Staubli VAL3: processList.pjx

--- processList.pjx ---
Parameters version=s7.2.1 stackSize=5000 millimeterUnit=true
Program file=delete.pgx
Program file=deleteAll.pgx
Program file=getCycle.pgx
Program file=getDefaultType.pgx
Program file=getLoaded.pgx
Program file=getLoop.pgx
Program file=getPath.pgx
Program file=getSize.pgx
Program file=increase.pgx
Program file=init.pgx
Program file=insertCycle.pgx
Program file=isFound.pgx
Program file=loadProcessList.pgx
Program file=loopMode.pgx
Program file=makeFile.pgx
Program file=save.pgx
Program file=selectType.pgx
Program file=setCycle.pgx
Program file=setDefaultType.pgx
Program file=setLoop.pgx
Data file=processList.dtx
Library alias=use path=Disk://kernel/userPage/userPage.pjx
Library alias=cycleStatus path=Disk://cycleStatus/cycleStatus.pjx
Library alias=saveData path=Disk://saveData/saveData.pjx
Library alias=language path=Disk://kernel/language/language.pjx
Library alias=saveCycle path=Disk://kernel/template/session/saveCycle/saveCycle.pjx autoload=false
Library alias=prog path=Disk://instruction/PROG/PROG.pjx
Library alias=OnEvent path=Disk://OnEvent/OnEvent.pjx

--- processList.dtx ---
num nFile
string sEvent
string sProcessList
string sType
string sWrite
bool bLoading
public bool bLoop = true

--- delete.pgx ---
public program delete(num x_nIndex, num x_nType)
begin
  // mutex for the loading
  setMutex(cycleStatus:bMutex)
  switch x_nType
    case 0
      // delete a program into the process list
      logMsg("[KERNEL] CYCLE:Delete the program: "+saveCycle:sLoadStart[x_nIndex]+" at the index: "+toString("",x_nIndex))
      if size(saveCycle:sLoadStart)>1
        delete(saveCycle:sLoadStart[x_nIndex])
        delete(saveCycle:nDoneStart[x_nIndex])
        delete(saveCycle:nTotalStart[x_nIndex])
      else
        saveCycle:sLoadStart[0]=""
        saveCycle:nDoneStart[0]=0
        saveCycle:nTotalStart[0]=0
      endIf
    break
    case 1
      logMsg("[KERNEL] CYCLE:Delete the program: "+saveCycle:sLoadProg[x_nIndex]+" at the index: "+toString("",x_nIndex))
      // delete a program into the process list
      if size(saveCycle:sLoadProg)>1
        delete(saveCycle:sLoadProg[x_nIndex])
        delete(saveCycle:nDoneCycle[x_nIndex])
        delete(saveCycle:nTotalCycle[x_nIndex])
      else
        saveCycle:sLoadProg[0]=""
        saveCycle:nDoneCycle[0]=0
        saveCycle:nTotalCycle[0]=0
      endIf
    break
    case 2
      logMsg("[KERNEL] CYCLE:Delete the program: "+saveCycle:sLoadEnd[x_nIndex]+" at the index: "+toString("",x_nIndex))
      // delete a program into the process list
      if size(saveCycle:sLoadEnd)>1
        delete(saveCycle:sLoadEnd[x_nIndex])
        delete(saveCycle:nDoneEnd[x_nIndex])
        delete(saveCycle:nTotalEnd[x_nIndex])
      else
        saveCycle:sLoadEnd[0]=""
        saveCycle:nDoneEnd[0]=0
        saveCycle:nTotalEnd[0]=0
      endIf
    break
  endSwitch
//  // in order to refresh the first program
//  if x_nIndex==0
//    cycleStatus:bProgLoad=false
//    cycleStatus:sProgLoad=""
//  endIf
  //
  cycleStatus:bMutex=false
end

--- deleteAll.pgx ---
public program deleteAll(num x_nType)
  local num i
  local num nSize[3]
begin
  // onEvent
  call OnEvent:OnCycleEvent(15)
  //
  logMsg("[KERNEL] CYCLE:Delete all the program..")
  call getSize(nSize,x_nType)
  for i=0 to (nSize-1)
    call delete(0,x_nType)
  endFor
  // reinit the buffer of all the program
  // cycleStatus:bInitMemory=true
end

--- getCycle.pgx ---
public program getCycle(string& x_sName[], num& x_nTotal[], num& x_nDone[], num x_nIndex, num x_nType)
begin
  // mutex it
  // setMutex
  setMutex(cycleStatus:bMutex)
  // get the cycle from the process LIST
  switch x_nType
    case 0
      if x_nIndex<size(saveCycle:sLoadStart)
        // ON START CYCLE
        x_sName=saveCycle:sLoadStart[x_nIndex]
        x_nTotal=saveCycle:nTotalStart[x_nIndex]
        x_nDone=saveCycle:nDoneStart[x_nIndex]
      endIf
    break
    case 1
      if x_nIndex<size(saveCycle:sLoadProg)
        // get the information about the actual process list
        x_sName=saveCycle:sLoadProg[x_nIndex]
        x_nTotal=saveCycle:nTotalCycle[x_nIndex]
        x_nDone=saveCycle:nDoneCycle[x_nIndex]
      endIf
    break
    case 2
      if x_nIndex<size(saveCycle:sLoadEnd)
        // ON END CYCLE
        x_sName=saveCycle:sLoadEnd[x_nIndex]
        x_nTotal=saveCycle:nTotalEnd[x_nIndex]
        x_nDone=saveCycle:nDoneEnd[x_nIndex]
      endIf
    break
  endSwitch
  // release
  cycleStatus:bMutex=false
end

--- getDefaultType.pgx ---
public program getDefaultType(num& x_nType[])
begin
  // get the process List
  // get the last type used
  x_nType=saveCycle:nType
end

--- getLoaded.pgx ---
public program getLoaded(string& x_sLoaded[])
// get the loaded processList
begin
  // give back the actual saveCycle
  x_sLoaded=saveCycle:libPath()
  // empty the string if is the default
  if find(x_sLoaded,"template/saveCycle")!=-1
    x_sLoaded=""
  endIf
  // give back the program
  call getPath(x_sLoaded)
end

--- getLoop.pgx ---
public program getLoop(bool& x_bLoop[])
begin
  // get the loop status
  x_bLoop=saveCycle:bLoop
end

--- getPath.pgx ---
program getPath(string& x_sType[])
  local num l_nPos
  local string l_sPath
  local num i
begin
  // get the TypePath
  l_sPath=x_sType
  do
    l_nPos=find(l_sPath,"/")
    if l_nPos==-1
      l_nPos=find(l_sPath,"\")
    endIf
    if l_nPos!=-1
      l_sPath=right(l_sPath,len(l_sPath)-l_nPos-1)
    endIf
  until l_nPos==-1
  // give BACK
  x_sType=l_sPath
end

--- getSize.pgx ---
public program getSize(num& x_nSize[], num x_nType)
begin
  // get the size of the Start list
  switch x_nType
    case 0
      // get the size of the Start list
      if saveCycle:sLoadStart!=""
        x_nSize=size(saveCycle:sLoadStart)
      else
        x_nSize=0
      endIf
    break
    case 1
      if saveCycle:sLoadProg!=""
        // get the size of the process list
        x_nSize=size(saveCycle:sLoadProg)
      else
        x_nSize=0
      endIf
    break
    case 2
      if saveCycle:sLoadEnd!=""
        // get the size of the End list
        x_nSize=size(saveCycle:sLoadEnd)
      else
        x_nSize=0
      endIf
    break
  endSwitch
end

--- increase.pgx ---
public program increase(num x_nType)
begin
  // increase the size plus 1
  switch x_nType
    case 0
      // START LIST
      saveCycle:nDoneStart[cycleStatus:nProg]=saveCycle:nDoneStart[cycleStatus:nProg]+1
    break
    case 1
      // PROCESS LIST
      saveCycle:nDoneCycle[0]=saveCycle:nDoneCycle[0]+1
    break
    case 2
      // END LIST
      saveCycle:nDoneEnd[cycleStatus:nProg]=saveCycle:nDoneEnd[cycleStatus:nProg]+1
    break
  endSwitch
end

--- init.pgx ---
public program init()
  local num i
begin
  // setMutex
  setMutex(cycleStatus:bMutex)
  // START CYCLE
  for i=0 to size(saveCycle:nDoneStart)-1
    saveCycle:nDoneStart[i]=0
  endFor
  // PROCESS LIST
  if saveCycle:bLoop
    for i=0 to size(saveCycle:nDoneCycle)-1
      saveCycle:nDoneCycle[i]=0
    endFor
  endIf
  // END CYCLE
  for i=0 to size(saveCycle:nDoneEnd)-1
    saveCycle:nDoneEnd[i]=0
  endFor
  //release
  cycleStatus:bMutex=false
end

--- insertCycle.pgx ---
public program insertCycle(num x_nIndex, string x_sName, num x_nTotal, num x_nDone, num x_nType)
  local num l_nIndex
begin
  // setMutex
  setMutex(cycleStatus:bMutex)
  // insert a cycle into the process list
  //
  // use x_nIndex -1 to use FIFO politc
  //
  if x_nIndex!=-1
    l_nIndex=x_nIndex
  else
    switch x_nType
      case 0
        // start List
        if size(saveCycle:sLoadStart)==1 and saveCycle:sLoadStart[0]==""
          l_nIndex=0
        else
          l_nIndex=(size(saveCycle:sLoadStart))
        endIf
      break
      case 1
        // production list
        if size(saveCycle:sLoadProg)==1 and saveCycle:sLoadProg[0]==""
          l_nIndex=0
        else
          l_nIndex=(size(saveCycle:sLoadProg))
        endIf
      break
      case 2
        // end List
        if size(saveCycle:sLoadEnd)==1 and saveCycle:sLoadEnd[0]==""
          l_nIndex=0
        else
          l_nIndex=(size(saveCycle:sLoadEnd))
        endIf
      break
    endSwitch
  endIf
  //
  // Val3 need to have at least 1 item into a vector so...
  //
  switch x_nType
    case 0
      // ON START CYCLE
      if (l_nIndex>0) and saveCycle:sLoadStart!=""
        insert(saveCycle:sLoadStart[l_nIndex])
        insert(saveCycle:nDoneStart[l_nIndex])
        insert(saveCycle:nTotalStart[l_nIndex])
      endIf
    break
    case 1
      // get the information about the actual process list
      if (l_nIndex>0) and saveCycle:sLoadProg!=""
        insert(saveCycle:sLoadProg[l_nIndex])
        insert(saveCycle:nDoneCycle[l_nIndex])
        insert(saveCycle:nTotalCycle[l_nIndex])
      endIf
    break
    case 2
      // ON END CYCLE
      if (l_nIndex>0) and saveCycle:sLoadEnd!=""
        insert(saveCycle:sLoadEnd[l_nIndex])
        insert(saveCycle:nDoneEnd[l_nIndex])
        insert(saveCycle:nTotalEnd[l_nIndex])
      endIf
    break
  endSwitch
  // set the cycle
  call setCycle(x_sName,x_nTotal,x_nDone,l_nIndex,x_nType)
  //release
  cycleStatus:bMutex=false
end

--- isFound.pgx ---
public program isFound(string& x_sName[], bool& x_bFound[])
  local num i
  local num j
  local num l_nSize[3]
  local string l_sString
  local num k
  local num l_nResult
  local string l_sEmpty
  local num l_nID
begin
  //
  // find if a program is inside the processList
  //
  x_bFound=false
  //
  // update
  //
  l_sEmpty=""
  call use:stringCopy(l_sEmpty,sProcessList)
  // check all
  call loadProcessList(l_nResult)
  // get the size of the three processList
  for i=0 to 2
    call getSize(l_nSize[i],i)
    // look in all the program
    for j=0 to max(l_nSize[i]-1,0)
      l_nID=0
      call getCycle(l_sString,l_nID,l_nID,j,i)
      if l_sString==x_sName
        x_bFound=true
        x_sName=l_sString
        return
      endIf
    endFor
  endFor
end

--- loadProcessList.pgx ---
public program loadProcessList(num& x_nResult[])
// load the process list
  local num i
  local string l_sMessage
  local string l_sMessage2
begin
  // setMutex
  setMutex(cycleStatus:bMutex)
  // load a different processList
  if cycleStatus:bCycle==false and cycleStatus:bSimulation==false
    //saveData:sPathPList+x_sProcess
    x_nResult=saveCycle:libLoad(saveData:sPathPList)
    delay(0)
    if saveData:bDebug and x_nResult!=0
      logMsg("[KERNEL] SETPROCESSLIST:Loading processList, CODE: "+toString("",x_nResult))
    endIf
    // check the result
    if x_nResult!=0
      // load the template and empty the list
      x_nResult=saveCycle:libLoad("kernel/template/session/saveCycle")
      delay(0)
      libDelete(saveData:sPathPList)
      saveCycle:libSave(saveData:sPathPList)
      // default process list has been charged
      call language:message(l_sMessage,-7)
      call language:message(l_sMessage2,97)
      popUpMsg(l_sMessage+"saveCycle... "+l_sMessage2)
    endIf
  else
    x_nResult=-1
  endIf
  //release
  cycleStatus:bMutex=false
end

--- loopMode.pgx ---
public program loopMode()
  local num i
  local string sSwapLoad
  local num nSwapTotal
  local num l_nSize
begin
  //  set the process list after one cycle done
  //
  //  the variable loadProg has to not be minus than 1 items
  //  THIS IS THE NO LOOP CODE
  //
  if !saveCycle:bLoop
    //
    call delete(0,1)
  else
    //
    //  LOOP MODE
    //
    call getSize(l_nSize,1)
    if cycleStatus:nProg<l_nSize-1
      // continue
      cycleStatus:nProg=cycleStatus:nProg+1
    else
      // REINIT
      for i=0 to l_nSize-1
        saveCycle:nDoneCycle[i]=0
      endFor
      cycleStatus:nProg=0
    endIf
  endIf
end

--- makeFile.pgx ---
public program makeFile()
  local num i
  local num j
  local num l_nSize[3]
  local num l_nType
  local string l_sProg
  local string l_sFill
  local string l_sMessage
  local string l_sEmpty
  local num l_nID
begin
  // check if the cycle is not running
  if cycleStatus:bCycle==false and cycleStatus:bSimulation==false
    // scan all the processList
    for i=0 to 2
      call getSize(l_nSize[i],i)
    endFor
    // check if the process List is empty
    if l_nSize[1]==0
      // show message
      call language:message(l_sMessage,91)
      popUpMsg(l_sMessage)
      // came back
      return
    endIf
    // scan it
    for l_nType=0 to 2
      //
      // init
      l_sEmpty=""
      call use:stringCopy(l_sEmpty,prog:sWrite)
      //
      switch l_nType
        case 0
          // START PROCESS LIST
          // open the file
          nFile=$fileOpen("start.txt","w")
        break
        case 1
          // PROCESS LIST
          // open the file
          nFile=$fileOpen("production.txt","w")
        break
        case 2
          // END PROCESS LIST
          // open the file
          nFile=$fileOpen("end.txt","w")
        break
      endSwitch
      // scan all the program
      if l_nSize[l_nType]>0
        for i=0 to (l_nSize[l_nType]-1)
          // get the cycle
          l_nID=0
          call getCycle(l_sProg,l_nID,l_nID,i,l_nType)
          // scan the system and save the process List
          // add the program name
          insert(prog:sWrite[0])
          insert(prog:sWrite[0])
          insert(prog:sWrite[0])
          // insert the program NAME
          for j=0 to len(l_sProg)-1
            l_sFill=l_sFill+"═"
          endFor
          prog:sWrite[0]="╔═════"+l_sFill+"╗"
          prog:sWrite[1]="║PROG "+l_sProg+"║"
          prog:sWrite[2]="╚═════"+l_sFill+"╝"
          // scan the program
          call use:timerDialog("Scanning the program: "+l_sProg+"# please wait...",0)
          l_nID=3
          call prog:scanning(l_sProg,0,l_nID,true)
          // write to the file
          $fileSet(nFile,prog:sWrite,size(prog:sWrite))
          // reset the sWrite buffer
          l_sEmpty=""
          call use:stringCopy(l_sEmpty,prog:sWrite)
          l_sFill=""
        endFor
        // save the file
        $fileClose(nFile)
      endIf
    endFor
  endIf
end

--- save.pgx ---
public program save()
// save the process list
  local num i
begin
  // setMutex
  setMutex(cycleStatus:bMutex)
  // save IT
  if saveCycle:libSave()!=0
    delay(0.5)
    i=saveCycle:libSave()
    if i!=0
      popUpMsg("libsave cycle error: "+toString("",i))
      logMsg("[KERNEL] CYCLE:Error saving cycle "+toString("",i))
    endIf
  endIf
  //release
  cycleStatus:bMutex=false
end

--- selectType.pgx ---
public program selectType()
  local string l_sMessage
  local num l_nIndex
  local string l_sEvent
  local num l_nDefault
  local num l_nKey
  local num i
begin
  // select the type of the process LIST
  call use:clear(0,13)
  call language:message(l_sMessage,191)
  call use:typeCenter(13,l_sMessage,40,true)
  call use:setSizeList(10,2,15,6)
  // TODO message
  call use:listcreate("")
  call use:listadd(sType)
  call getDefaultType(l_nDefault)
  call use:selectNewField(l_nDefault,0,0)
  // select the Item
  do
    l_nKey=get()
    call use:listevent(l_nKey,l_nIndex,l_sEvent)
    // search for a key
  until l_nKey==270 or l_nKey==255
  if l_nKey==270
    call setDefaultType(l_nIndex)
    use:bUseRefresh=true
  endIf
  //
end

--- setCycle.pgx ---
public program setCycle(string x_sName, num x_nTotal, num x_nDone, num x_nIndex, num x_nType)
begin
  // insert one cycle in the processLIST
  switch x_nType
    case 0
      // ON START CYCLE
      logMsg("[KERNEL] CYCLE:Insert the program: "+x_sName+" at the position: "+toString("",x_nIndex))
      saveCycle:sLoadStart[x_nIndex]=x_sName
      saveCycle:nTotalStart[x_nIndex]=x_nTotal
      saveCycle:nDoneStart[x_nIndex]=x_nDone
    break
    case 1
      // get the information about the actual process list
      logMsg("[KERNEL] CYCLE:Insert the program: "+x_sName+" at the position: "+toString("",x_nIndex))
      saveCycle:sLoadProg[x_nIndex]=x_sName
      saveCycle:nTotalCycle[x_nIndex]=x_nTotal
      saveCycle:nDoneCycle[x_nIndex]=x_nDone
    break
    case 2
      // ON END CYCLE
      logMsg("[KERNEL] CYCLE:Insert the program: "+x_sName+" at the position: "+toString("",x_nIndex))
      saveCycle:sLoadEnd[x_nIndex]=x_sName
      saveCycle:nTotalEnd[x_nIndex]=x_nTotal
      saveCycle:nDoneEnd[x_nIndex]=x_nDone
    break
  endSwitch
end

--- setDefaultType.pgx ---
public program setDefaultType(num& x_nType[])
begin
  // set the last type used
  saveCycle:nType=x_nType
end

--- setLoop.pgx ---
public program setLoop(bool x_bLoop)
  local string loop
begin
  // set the loop to ON OFF
  if x_bLoop
    loop="ON"
  else
    loop="OFF"
  endIf
  // set cycle LIST
  logMsg("[KERNEL] CYCLE:Set the loop mode to: "+loop)
  saveCycle:bLoop=x_bLoop
end
